{attribute 'TcGenerated'}
{attribute 'no-analysis'}
{attribute 'linkalways'}
// This function has been automatically generated from the project information.
VAR_GLOBAL CONSTANT
	{attribute 'const_non_replaced'}
	stLibVersion_OPC_UA_client : ST_LibVersion := (iMajor := 0, iMinor := 1, iBuild := 0, iRevision := 0, nFlags := 0, sVersion := '0.1');
END_VAR

(* stored: Version 1.1.0.1, ProductVersion 3.1.4024.9
   GVL Global_Version: Id {8ac0f2fa-6765-4c0e-aebf-c566c5b2c5cf} *)
